// TIA Portal V15.1 export
// export: Created 2024-05-17T05:38:44.7001503Z, ExportSetting WithDefaults, DisplayName Totally Integrated Automation Portal, DisplayVersion V15.1 Update 5, DisplayName TIA Portal Openness, DisplayVersion V15.1 Update 5, DisplayName SINAMICS Startdrive Advanced, DisplayVersion V15.1, DisplayName G130, G150, S120, S150, SINAMICS MV, S210, DisplayVersion V15.1, DisplayName G110M, G120, G120C, G120D, G120P, DisplayVersion V15.1, DisplayName STEP 7 Professional, DisplayVersion V15.1 Update 5, DisplayName STEP 7 Safety, DisplayVersion V15.1, DisplayName WinCC Professional, DisplayVersion V15.1 Update 5, DisplayName SIMATIC Visualization Architect, DisplayVersion V15.1
FUNCTION_BLOCK "LGBProdInfo"   // FB6702, FBD
TITLE = LGBProdInfo
{ S7_Optimized_Access := 'TRUE' }
VERSION : 0.1
// stored: AutoNumber false, IsIECCheckEnabled false, IsRetainMemResEnabled false, MemoryReserve 100, SetENOAutomatically False, UDAEnableTagReadback false
   VAR_INPUT
      I_ConfigProdSpeed { ExternalAccessible := 'False'; ExternalVisible := 'False'; ExternalWritable := 'False'} : "ProdSpeedConfig";   // Config
      I_ConfigProdStartStop { ExternalAccessible := 'False'; ExternalVisible := 'False'; ExternalWritable := 'False'} : "ProdStartStopConfig";   // Config
      I_ConfigLineFeed { ExternalAccessible := 'False'; ExternalVisible := 'False'; ExternalWritable := 'False'} : "LineFeedConfig";   // Config
      I_ConfigShiftRegLine { ExternalAccessible := 'False'; ExternalVisible := 'False'; ExternalWritable := 'False'} : "ShiftRegLineConfig";   // Output Word / Config
   END_VAR
   VAR_IN_OUT
      H_GBProdInfo : "H_GBProdInfo";   // Animation
   END_VAR
BEGIN

REGION Network 1: **** 4.6 - Machine status - Indications **** Animation
   // Animation Word 1
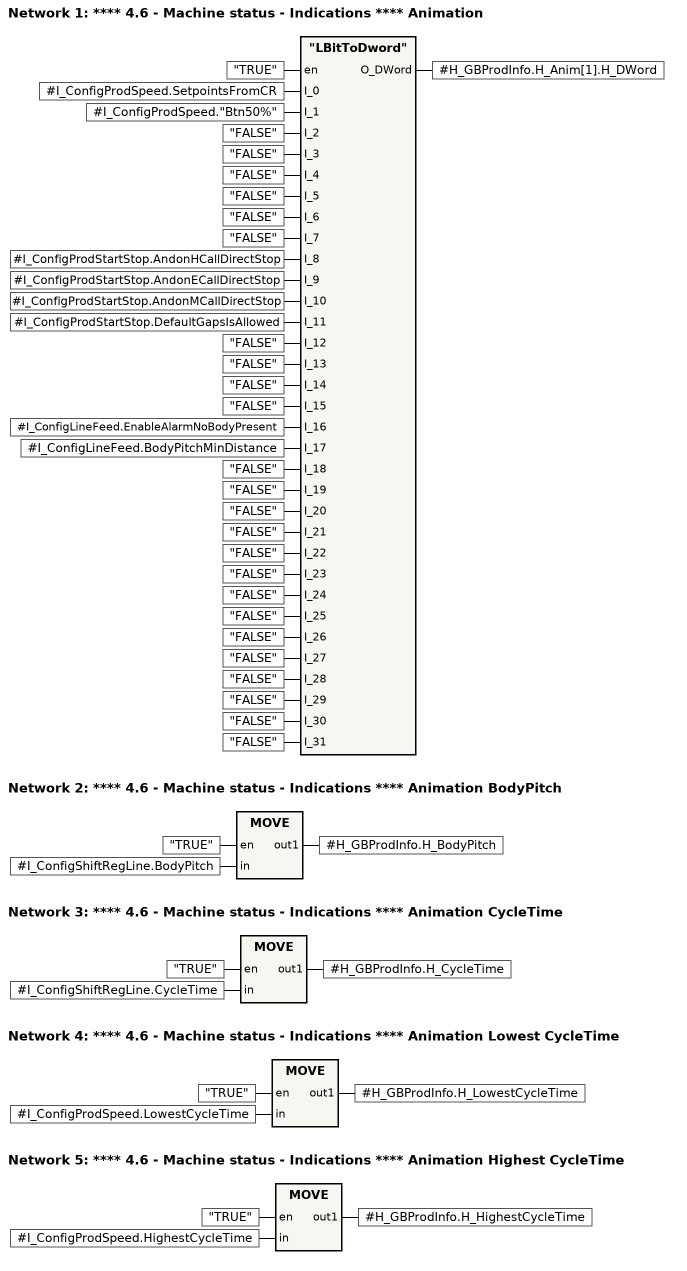
   IF "TRUE" THEN
       "LBitToDword"(I_0 := #I_ConfigProdSpeed.SetpointsFromCR,
                     I_1 := #I_ConfigProdSpeed."Btn50%",
                     I_2 := "FALSE",
                     I_3 := "FALSE",
                     I_4 := "FALSE",
                     I_5 := "FALSE",
                     I_6 := "FALSE",
                     I_7 := "FALSE",
                     I_8 := #I_ConfigProdStartStop.AndonHCallDirectStop,
                     I_9 := #I_ConfigProdStartStop.AndonECallDirectStop,
                     I_10 := #I_ConfigProdStartStop.AndonMCallDirectStop,
                     I_11 := #I_ConfigProdStartStop.DefaultGapsIsAllowed,
                     I_12 := "FALSE",
                     I_13 := "FALSE",
                     I_14 := "FALSE",
                     I_15 := "FALSE",
                     I_16 := #I_ConfigLineFeed.EnableAlarmNoBodyPresent,
                     I_17 := #I_ConfigLineFeed.BodyPitchMinDistance,
                     I_18 := "FALSE",
                     I_19 := "FALSE",
                     I_20 := "FALSE",
                     I_21 := "FALSE",
                     I_22 := "FALSE",
                     I_23 := "FALSE",
                     I_24 := "FALSE",
                     I_25 := "FALSE",
                     I_26 := "FALSE",
                     I_27 := "FALSE",
                     I_28 := "FALSE",
                     I_29 := "FALSE",
                     I_30 := "FALSE",
                     I_31 := "FALSE",
                     O_DWord => #H_GBProdInfo.H_Anim[1].H_DWord);
   END_IF;
END_REGION

REGION Network 2: **** 4.6 - Machine status - Indications **** Animation BodyPitch
   IF "TRUE" THEN #H_GBProdInfo.H_BodyPitch := #I_ConfigShiftRegLine.BodyPitch; END_IF;
END_REGION

REGION Network 3: **** 4.6 - Machine status - Indications **** Animation CycleTime
   IF "TRUE" THEN #H_GBProdInfo.H_CycleTime := #I_ConfigShiftRegLine.CycleTime; END_IF;
END_REGION

REGION Network 4: **** 4.6 - Machine status - Indications **** Animation Lowest CycleTime
   IF "TRUE" THEN #H_GBProdInfo.H_LowestCycleTime := #I_ConfigProdSpeed.LowestCycleTime; END_IF;
END_REGION

REGION Network 5: **** 4.6 - Machine status - Indications **** Animation Highest CycleTime
   IF "TRUE" THEN #H_GBProdInfo.H_HighestCycleTime := #I_ConfigProdSpeed.HighestCycleTime; END_IF;
END_REGION
END_FUNCTION_BLOCK
